PROGRAM Process
VAR
	Tramp_FB: Tramp;
END_VAR

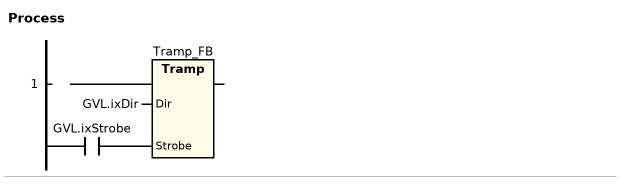
// NETWORK 1
Tramp_FB(Dir := GVL.ixDir, Strobe := GVL.ixStrobe); // Tramp

END_PROGRAM

(* stored: Version 1.1.0.1, ProductVersion 3.1.4024.12
   POU Process: Id {59590995-2b72-4d4f-a7f9-4ba974045ea5}, SpecialFunc None *)
